(* IEC 61131-3 sources: BuT/takt-lang/tests/data/st/probes, 7 files *)

(* ---- probe_array.st ---- *)
(* Проба: ARRAY в VAR блока FB. *)
FUNCTION_BLOCK Demo
VAR
    data : ARRAY [0..3] OF USINT;
    i : USINT := 0;
END_VAR
    data[0] := 7;
    data[1] := data[0] + 1;
END_FUNCTION_BLOCK

(* ---- probe_at.st ---- *)
(* П8. VAR_GLOBAL ... AT %IX + VAR_EXTERNAL в FB.
   Подтверждает форму 0041-05 (AddressMap → AT %...). *)
VAR_GLOBAL
    Button AT %IX256.0 : BOOL;
    Lamp   AT %QX256.1 : BOOL;
END_VAR

FUNCTION_BLOCK Demo
VAR_EXTERNAL
    Button : BOOL;
    Lamp : BOOL;
END_VAR
    Lamp := Button;
END_FUNCTION_BLOCK

(* ---- probe_enum.st ---- *)
(* П4. Перечислимый TYPE с явными значениями.
   Решает T13 (0041-02): прямое отображение enum Takt → TYPE, или откат
   Option C (USINT + VAR_GLOBAL CONSTANT). *)
TYPE
    Floor : (Bottom := 80, Top);
END_TYPE

FUNCTION_BLOCK Demo
VAR
    f : Floor := Bottom;
END_VAR
    IF f = Bottom THEN
        f := Top;
    END_IF;
END_FUNCTION_BLOCK

(* ---- probe_fb.st ---- *)
(* П2. Голый FUNCTION_BLOCK без CONFIGURATION.
   Ключевая проба: принимает ли iec2c отдельный блок, или требует полной
   программы для ПЛК. От исхода зависит, обязан ли генератор эмитить
   CONFIGURATION (флаг --st-configuration). *)
FUNCTION_BLOCK Demo
VAR
    state : USINT := 0;
    count : USINT := 0;
END_VAR
    CASE state OF
        0:
            count := count + 1;
            IF count >= 3 THEN
                state := 1;
            END_IF;
        1:
            count := 0;
    END_CASE;
END_FUNCTION_BLOCK

(* ---- probe_full.st ---- *)
(* П3. Полная обёртка: CONFIGURATION / RESOURCE / TASK / PROGRAM.
   Форма, которую генератор обязан эмитить, если П2 красная. *)
FUNCTION_BLOCK Demo
VAR
    state : USINT := 0;
    count : USINT := 0;
END_VAR
    CASE state OF
        0:
            count := count + 1;
        1:
            count := 0;
    END_CASE;
END_FUNCTION_BLOCK

PROGRAM Main
VAR
    inst : Demo;
END_VAR
    inst();
END_PROGRAM

CONFIGURATION Config0
    RESOURCE Res0 ON PLC
        TASK Tick(INTERVAL := T#100ms, PRIORITY := 0);
        PROGRAM Inst0 WITH Tick : Main;
    END_RESOURCE
END_CONFIGURATION

(* ---- probe_inout.st ---- *)
(* П7. VAR_IN_OUT и вызов FB из FB.
   Решает О1 (0041-03): как под-FB видят переменные корня. Самый рискованный
   вопрос семантики фичи — в Takt композиция `A | B` даёт под-моделям доступ к
   портам корня в том же такте. *)
FUNCTION_BLOCK Child
VAR_IN_OUT
    shared : USINT;
END_VAR
VAR
    state : USINT := 0;
END_VAR
    shared := shared + 1;
END_FUNCTION_BLOCK

FUNCTION_BLOCK Parent
VAR
    value : USINT := 0;
    kid : Child;
END_VAR
    kid(shared := value);
END_FUNCTION_BLOCK

(* ---- probe_lreal.st ---- *)
(* Проба: LREAL - 64-битное вещественное.
   Симулятор Takt считает в f64, поэтому LREAL, а не REAL. *)
FUNCTION_BLOCK Demo
VAR
    x : LREAL := 0.5;
END_VAR
    x := x * 2.0;
END_FUNCTION_BLOCK
